// TwinCAT 3 PLC project ArucoScanner
// ProgramVersion: 3.1.4024.0
// libraries:
//   Tc2_Standard, * (Beckhoff Automation GmbH)
//   Tc2_System, * (Beckhoff Automation GmbH)
//   Tc3_Module, * (Beckhoff Automation GmbH)
//   Tc3_Vision, * (Beckhoff Automation GmbH)
// project tree:
//   DUTs/ ImageDataTest.TcDUT
//   / PlcTask.TcTTO
//   POUs/ MAIN.TcPOU

CONFIGURATION ArucoScanner
    RESOURCE PLC ON TwinCAT3
        TASK PlcTask(INTERVAL := T#10ms, PRIORITY := 20);
        PROGRAM MAIN WITH PlcTask : MAIN;
    END_RESOURCE
END_CONFIGURATION

// ---- DUTs/ImageDataTest.TcDUT
TYPE ImageDataTest :
STRUCT
    data : ARRAY [0..307200] OF BYTE; // for a 640x480 grayscale image
END_STRUCT
END_TYPE

// ---- POUs/MAIN.TcPOU
PROGRAM MAIN
VAR
	hr 							: HRESULT;
	fbCamera 					: FB_VN_SimpleCameraControl;
	eState 						: ETcVnCameraState;
	ipImageIn		    		: ITcVnImage;
	ipProcessedImage    		: ITcVnImage;
	ipImageInDisplay 			: ITcVnDisplayableImage;
	ipProcessedImageToDisplay 	: ITcVnDisplayableImage;
END_VAR

eState := fbCamera.GetState();

IF eState = TCVN_CS_ERROR THEN
	hr := fbCamera.Reset();
	
	ELSIF eState < TCVN_CS_ACQUIRING THEN
		hr := fbCamera.StartAcquisition();
		
		ELSIF eState = TCVN_CS_ACQUIRING THEN
			hr := fbCamera.GetCurrentImage(ipImageIn);
			
			IF SUCCEEDED(hr) AND ipImageIn <> 0 THEN
				hr := F_VN_Threshold(
				ipSrcImage      :=  ipImageIn,
				ipDestImage     :=  ipProcessedImage,
				fThreshold      :=  128, // half value range: (2^8)/2=128
				fMaxValue       :=  255, // max value of 8-bit image: (2^8)-1=255
				eThresholdType  :=  TCVN_TT_BINARY,
				hrPrev          :=  hr
			);
			hr := F_VN_TransformIntoDisplayableImage(ipProcessedImage, ipProcessedImageToDisplay, hr); //threshold Image
			hr := F_VN_TransformIntoDisplayableImage(ipImageIn, ipImageInDisplay, hr);        // raw image
			END_IF
END_IF

END_PROGRAM
